INTERFACE I_AsyncCommand extends I_Command

METHOD PUBLIC Abort
VAR_INPUT
END_VAR
END_METHOD

PROPERTY PUBLIC Busy : BOOL
GET
END_GET
END_PROPERTY

METHOD PUBLIC CyclicCall
VAR_INPUT
END_VAR
END_METHOD

PROPERTY PUBLIC Done : BOOL
GET
END_GET
END_PROPERTY

PROPERTY PUBLIC Error : BOOL
GET
END_GET
END_PROPERTY

PROPERTY PUBLIC ErrorId : UDINT
GET
END_GET
END_PROPERTY

END_INTERFACE

(* stored: Version 1.1.0.1, ProductVersion 3.1.4024.12
   Itf I_AsyncCommand: Id {c4e7ece3-ea49-01d2-328a-293a02955a0c}
   Method Abort: Id {700675eb-2a25-03f2-1387-a09f575adbca}
   Property Busy: Id {78824515-2a7b-0a05-18ea-f369d6766c82}
   Get Get: Id {d8c1f492-e1dc-0704-234f-3f9aa6d3dd6a}
   Method CyclicCall: Id {ec20b47b-6ab9-0741-1cf0-399a48d981ee}
   Property Done: Id {d48ed198-8c1b-0c01-05ae-20a41189aecf}
   Get Get: Id {2b3edc4c-c04d-0be6-2d58-5917d849262f}
   Property Error: Id {da914352-cf18-0c94-038e-4dd8d16d3749}
   Get Get: Id {0cb3b006-02c3-0916-244d-a10f89db41e9}
   Property ErrorId: Id {68c495e6-1d0f-09d6-18ae-e5af92e8a271}
   Get Get: Id {e8af2139-cfb9-0758-1844-a5b2163af0a2} *)
